PROGRAM MAIN
VAR
	b_groen_h 	: BOOL;
	b_oranje_h 	: BOOL;
	b_rood_h 	: BOOL;
	b_rood_v 	: BOOL;
	b_groen_v 	: BOOL;
	b_oranje_v 	: BOOL;
END_VAR

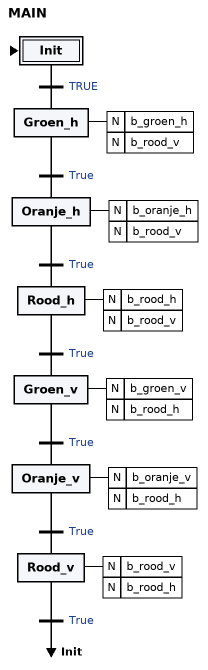
INITIAL_STEP Init:
END_STEP
TRANSITION FROM Init TO Groen_h
    := TRUE;
END_TRANSITION
STEP Groen_h:  // min time t#1000ms
    b_groen_h(N);
    b_rood_v(N);
END_STEP
TRANSITION FROM Groen_h TO Oranje_h
    := True;
END_TRANSITION
STEP Oranje_h:  // min time t#1000ms
    b_oranje_h(N);
    b_rood_v(N);
END_STEP
TRANSITION FROM Oranje_h TO Rood_h
    := True;
END_TRANSITION
STEP Rood_h:  // min time t#1000ms
    b_rood_h(N);
    b_rood_v(N);
END_STEP
TRANSITION FROM Rood_h TO Groen_v
    := True;
END_TRANSITION
STEP Groen_v:  // min time t#1000ms
    b_groen_v(N);
    b_rood_h(N);
END_STEP
TRANSITION FROM Groen_v TO Oranje_v
    := True;
END_TRANSITION
STEP Oranje_v:  // min time t#1000ms
    b_oranje_v(N);
    b_rood_h(N);
END_STEP
TRANSITION FROM Oranje_v TO Rood_v
    := True;
END_TRANSITION
STEP Rood_v:  // min time t#1000ms
    b_rood_v(N);
    b_rood_h(N);
END_STEP
TRANSITION FROM Rood_v TO Init
    := True;
END_TRANSITION

END_PROGRAM

(* stored: Version 1.1.0.1, ProductVersion 3.1.4024.12
   POU MAIN: Id {75926967-c251-4ba9-951d-93d020aa9aeb}, SpecialFunc None *)
